FUNCTION updateEventWithTimestamp : DATE_AND_TIME
VAR_INPUT
	stEvent : REFERENCE TO ST_Event;
END_VAR
VAR
	fbSystemTime : GETSYSTEMTIME;
    timeAsFileTime : T_FILETIME;
END_VAR

fbSystemTime(timeLoDW => timeAsFileTime.dwLowDateTime, timeHiDW => timeAsFileTime.dwHighDateTime);
stEvent.timestamp := FILETIME_TO_DT(timeAsFileTime);

END_FUNCTION

(* stored: Version 1.1.0.1
   POU updateEventWithTimestamp: Id {4c121f0d-0f57-4a74-8c03-6872026d6797}, SpecialFunc None *)
